% RSLogix 500 project P8 - PID Substitution Logic.RSS, saved by version 8.30.00.16 %
PROJECT "P8"    % processor: Bul.1763 MicroLogix 1100 Series B %

PROGRAM FILES
  LAD 2 "MAIN"  12 rungs

DATA FILES
  O0 OUTPUT  4 elements
  I1 INPUT  6 elements
  S2 STATUS  66 elements
  B3 BINARY  1 elements
  T4 TIMER  2 elements
  C5 COUNTER  1 elements
  R6 CONTROL  1 elements
  N7 INTEGER  3 elements
  F8 FLOAT  1 elements

LADDER 2 "MAIN"
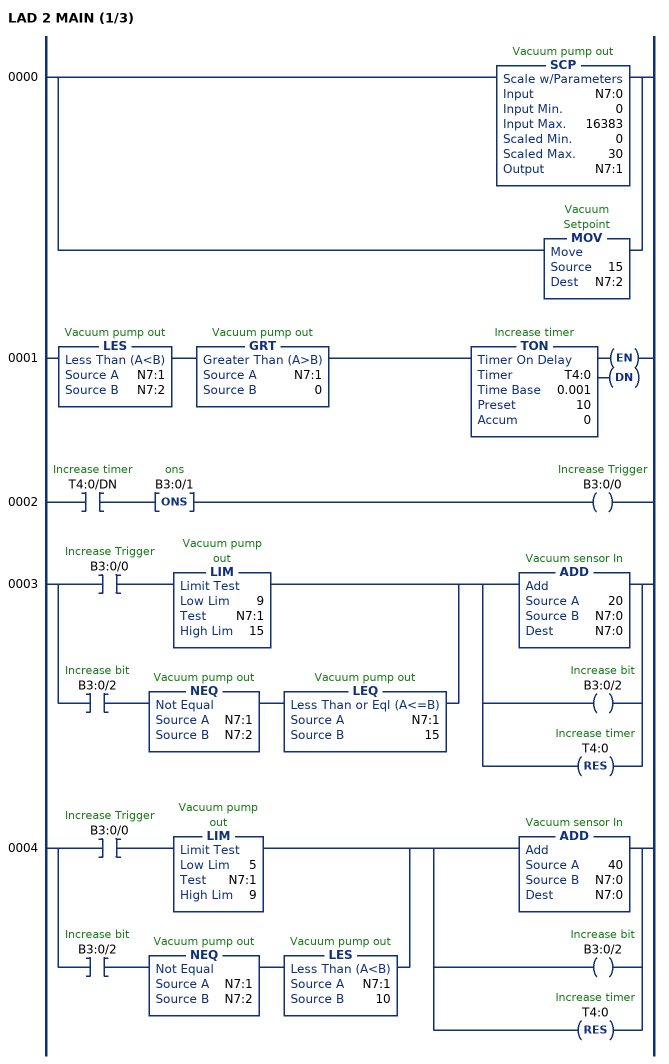
% Rung: 0 %
SOR BST SCP N7:0 0 16383 0 30 N7:1 NXB MOV 15 N7:2 BND EOR
%   N7:0  "Vacuum sensor In" %
%   N7:1  "Vacuum pump out" %
%   N7:2  "Vacuum Setpoint" %
% Rung: 1 %
SOR LES N7:1 N7:2 GRT N7:1 0 TON T4:0 0.001 10 0 EOR
%   N7:1  "Vacuum pump out" %
%   N7:2  "Vacuum Setpoint" %
%   T4:0  "Increase timer" %
% Rung: 2 %
SOR XIC T4:0/DN ONS B3:0/1 OTE B3:0/0 EOR
%   T4:0  "Increase timer" %
%   B3:0/1  "ons" %
%   B3:0/0  "Increase Trigger" %
% Rung: 3 %
SOR BST XIC B3:0/0 LIM 9 N7:1 15 NXB XIC B3:0/2 NEQ N7:1 N7:2 LEQ N7:1 15 BND BST ADD 20 N7:0 N7:0 NXB OTE B3:0/2 NXB RES T4:0 BND EOR
%   B3:0/0  "Increase Trigger" %
%   N7:1  "Vacuum pump out" %
%   B3:0/2  "Increase bit" %
%   N7:2  "Vacuum Setpoint" %
%   N7:0  "Vacuum sensor In" %
%   T4:0  "Increase timer" %
% Rung: 4 %
SOR BST XIC B3:0/0 LIM 5 N7:1 9 NXB XIC B3:0/2 NEQ N7:1 N7:2 LES N7:1 10 BND BST ADD 40 N7:0 N7:0 NXB OTE B3:0/2 NXB RES T4:0 BND EOR
%   B3:0/0  "Increase Trigger" %
%   N7:1  "Vacuum pump out" %
%   B3:0/2  "Increase bit" %
%   N7:2  "Vacuum Setpoint" %
%   N7:0  "Vacuum sensor In" %
%   T4:0  "Increase timer" %

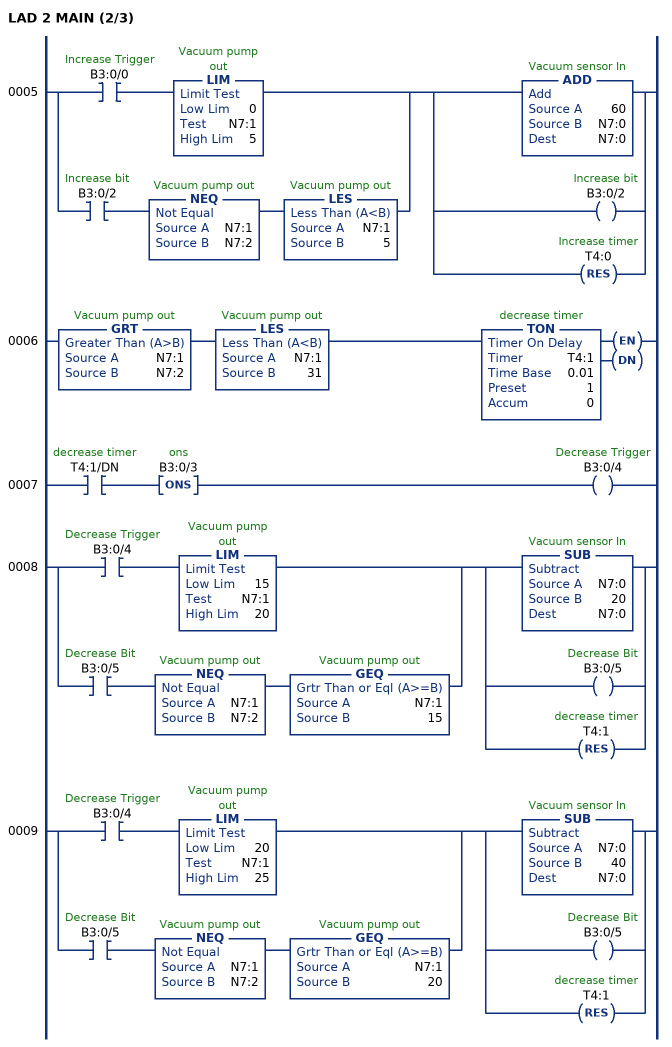
% Rung: 5 %
SOR BST XIC B3:0/0 LIM 0 N7:1 5 NXB XIC B3:0/2 NEQ N7:1 N7:2 LES N7:1 5 BND BST ADD 60 N7:0 N7:0 NXB OTE B3:0/2 NXB RES T4:0 BND EOR
%   B3:0/0  "Increase Trigger" %
%   N7:1  "Vacuum pump out" %
%   B3:0/2  "Increase bit" %
%   N7:2  "Vacuum Setpoint" %
%   N7:0  "Vacuum sensor In" %
%   T4:0  "Increase timer" %
% Rung: 6 %
SOR GRT N7:1 N7:2 LES N7:1 31 TON T4:1 0.01 1 0 EOR
%   N7:1  "Vacuum pump out" %
%   N7:2  "Vacuum Setpoint" %
%   T4:1  "decrease timer" %
% Rung: 7 %
SOR XIC T4:1/DN ONS B3:0/3 OTE B3:0/4 EOR
%   T4:1  "decrease timer" %
%   B3:0/3  "ons" %
%   B3:0/4  "Decrease Trigger" %
% Rung: 8 %
SOR BST XIC B3:0/4 LIM 15 N7:1 20 NXB XIC B3:0/5 NEQ N7:1 N7:2 GEQ N7:1 15 BND BST SUB N7:0 20 N7:0 NXB OTE B3:0/5 NXB RES T4:1 BND EOR
%   B3:0/4  "Decrease Trigger" %
%   N7:1  "Vacuum pump out" %
%   B3:0/5  "Decrease Bit" %
%   N7:2  "Vacuum Setpoint" %
%   N7:0  "Vacuum sensor In" %
%   T4:1  "decrease timer" %
% Rung: 9 %
SOR BST XIC B3:0/4 LIM 20 N7:1 25 NXB XIC B3:0/5 NEQ N7:1 N7:2 GEQ N7:1 20 BND BST SUB N7:0 40 N7:0 NXB OTE B3:0/5 NXB RES T4:1 BND EOR
%   B3:0/4  "Decrease Trigger" %
%   N7:1  "Vacuum pump out" %
%   B3:0/5  "Decrease Bit" %
%   N7:2  "Vacuum Setpoint" %
%   N7:0  "Vacuum sensor In" %
%   T4:1  "decrease timer" %

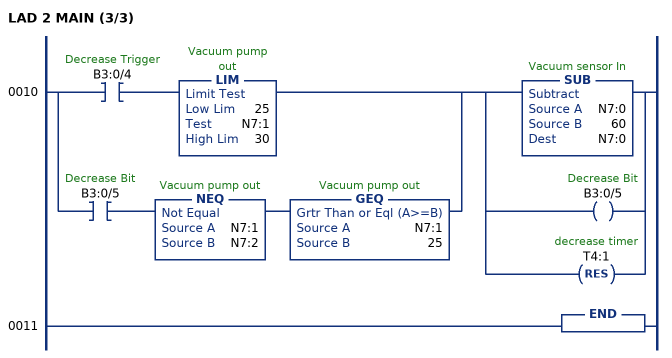
% Rung: 10 %
SOR BST XIC B3:0/4 LIM 25 N7:1 30 NXB XIC B3:0/5 NEQ N7:1 N7:2 GEQ N7:1 25 BND BST SUB N7:0 60 N7:0 NXB OTE B3:0/5 NXB RES T4:1 BND EOR
%   B3:0/4  "Decrease Trigger" %
%   N7:1  "Vacuum pump out" %
%   B3:0/5  "Decrease Bit" %
%   N7:2  "Vacuum Setpoint" %
%   N7:0  "Vacuum sensor In" %
%   T4:1  "decrease timer" %
% Rung: 11 %
SOR END EOR

OTHER DOCUMENTED ADDRESSES
  U:3  "I/O"

DATA TABLE (non-zero values as saved)
DATA T4
% .PRE .ACC %
% T4:0 % 10 0
% T4:1 % 1 0
